// TIA Portal V21 export
TYPE "OBJ_Encoder_SICK_AFM60_V105_Type"
   STRUCT
      IO : Struct
         IN { S7_SetPoint := 'True'} : "OBJ_IODevice_IN_SICK_AFM60_Tel81_V105_Type";
         OUT { S7_SetPoint := 'True'} : "OBJ_IODevice_OUT_SICK_AFM60_Tel81_V105_Type";
         App { ExternalAccessible := 'False'; ExternalVisible := 'False'; ExternalWritable := 'False'} : Struct
            Req_Writing_Preset : Bool;
            P_Write_Done : Bool;
            P_Write_Busy : Bool;
            P_Write_Error : Bool;
            P_Write_Req : Bool;
            P_Write_Status : DWord;
            Write_Requested : Bool;
            Ton { S7_SetPoint := 'True'} : IEC_TIMER;
            Toff { S7_SetPoint := 'True'} : IEC_TIMER;
            abil_zero { S7_SetPoint := 'True'} : Bool;
            set_zero : Bool;
         END_STRUCT;
      END_STRUCT;
      Data : Struct
         HMI : Struct
            "b_PB Zero" : Bool;
            "r_Actual Pos" : Real;   // Actual position (Real)
         END_STRUCT;
         CFG : Struct
            b_REQ_Offset : Bool;   // azzeramento al preset della conf. hw.
            b_REQ_SetUp : Bool;   // calcolo K factor
            r_ZeroOffset { S7_SetPoint := 'True'} : Real := 600000.0;   // Impulsi
            r_Cnt_Turn { S7_SetPoint := 'True'} : Real := 4096.0;   // Impulsi/giro
            r_LU_Turn { S7_SetPoint := 'True'} : Real := 1.0;   // mm/giro encoder
            r_K_Factor { S7_SetPoint := 'True'} : Real := 2048.0;   // fattore di conversione Impulsi/mm
            r_EncoderMaxCount { S7_SetPoint := 'True'} : Real;   // Impulsi
         END_STRUCT;
         SUP : Struct
            r_Raw_Val : Real;   // Raw Value from Encoder
         END_STRUCT;
      END_STRUCT;
      App { ExternalAccessible := 'False'; ExternalVisible := 'False'; ExternalWritable := 'False'} : Struct
         Ton { S7_SetPoint := 'True'} : IEC_TIMER;
      END_STRUCT;
   END_STRUCT;
END_TYPE
